FUNCTION_BLOCK BLINK
VAR_INPUT
	ENABLE: BOOL;
END_VAR
VAR_OUTPUT
	OUT: BOOL;
END_VAR
VAR
	TIMELOW: INT;
	TIMEHIGH: INT;
	T37: TON;
	T38: TOF;
	TEMP1: BOOL;
END_VAR

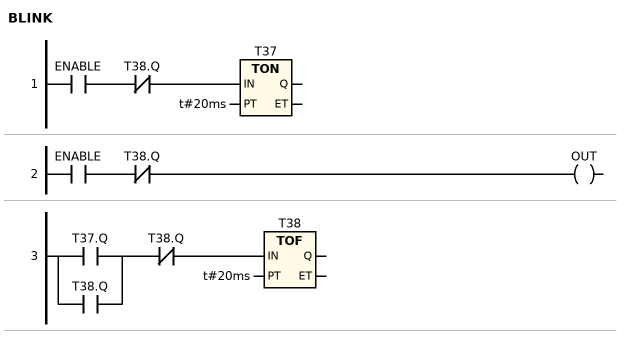
// NETWORK 1
T37(IN := ENABLE AND NOT T38.Q, PT := t#20ms); // TON

// NETWORK 2
OUT := ENABLE AND NOT T38.Q;

// NETWORK 3
T38(IN := (T37.Q OR T38.Q) AND NOT T38.Q, PT := t#20ms); // TOF

END_FUNCTION_BLOCK

(* stored: Version 1.1.0.1, ProductVersion 3.1.4024.12
   POU BLINK: Id {58f603e1-389b-44da-93f8-0a46e42efe1f}, SpecialFunc None *)
